Universal Robots PolyScope program: realtime.urp

Program realtime (installation=default directory=/programs/usbdisk/SanDiskSecureAccess createdIn=3.11.0.82155 lastSavedIn=3.11.0.82155 robotSerialNumber=2019301834)
Calibrated DH parameters: a=[0.000053, -0.592624, -0.100129, 0.000046, 0.000029, 0]; d=[0.128189, -50.911316, -326.675288, 377.750867, 0.115525, 0.092266]; alpha=[1.570692, -0.003019, -0.001489, 1.569354, -1.572015, 0]; deltaTheta=[-0.000027, 0.25377, 1.140819, -1.394601, -0.000039, 0.000039]
InitVariablesNode variables(variable(name=primed, expression=False))
Robot Program (runOnlyOnce=false)
  If primed≟ True
    Script: servoj(target,0,0,0.008, 0.2, 100)
  Else 
    Script: socket_open("192.168.1.37", 12347, "socket_10")
    Script: socket_send_line("ping", "socket_10")
    rawTarget := socket_read_ascii_float(6, "socket_10", 0)
    target := [rawTarget[1],rawTarget[2],rawTarget[3],rawTarget[4],rawTarget[5],rawTarget[6]]
    MoveJ speed 60 deg/s, acceleration 80 deg/s^2 (useActiveTCP=true)
      Waypoint Waypoint (Variable): variable=target
    primed := True
Thread Thread_1 (runOnlyOnce=false)
  If primed≟ True
    Script: socket_send_line("ping", "socket_10")
    rawTarget := socket_read_ascii_float(6, "socket_10", 0)
    target := [rawTarget[1],rawTarget[2],rawTarget[3],rawTarget[4],rawTarget[5],rawTarget[6]]
